{attribute 'linkalways'} 
{attribute 'no_explicit_call' := 'This FB is a CLASS and must be accessed using methods or properties'}
{attribute 'enable_dynamic_creation'}
FUNCTION_BLOCK FINAL ABS_LREAL EXTENDS Node
VAR
	in : _LREAL(0.0);
	out : _LREAL(0.0);
END_VAR

METHOD PUBLIC Clone : I_Node
VAR
	pNode : POINTER TO ABS_LREAL;
END_VAR
pNode := __NEW(ABS_LREAL);
Clone := pNode^;
END_METHOD

METHOD FB_init : BOOL
VAR_INPUT
	bInitRetains : BOOL; // if TRUE, the retain variables are initialized (warm start / cold start)
	bInCopyCode : BOOL;  // if TRUE, the instance afterwards gets moved into the copy code (online change)
END_VAR
AddInput('in',THIS^.in);
AddOutput('out', THIS^.out);
END_METHOD

METHOD PROTECTED OnExecute
VAR
END_VAR
out.Value := ABS(in.Value);
END_METHOD

END_FUNCTION_BLOCK

(* stored: Version 1.1.0.1, ProductVersion 3.1.4024.15
   POU ABS_LREAL: Id {fcfff1c8-c9fc-481f-9a21-d791f9ec23e7}, SpecialFunc None
   Folder Constructor: Id {4858954c-d1e2-43ab-ae90-4c9653a1e7e4}
   Method Clone: Id {40a193b8-4659-4bf7-b301-085966454971}
   Method FB_init: Id {009d6482-ae35-4f6b-b048-c159b2f8ea4b}
   Method OnExecute: Id {8f603b14-bb3e-443e-8ed1-810377d9415f} *)
